Staubli VAL3: FibraHSI.pjx

--- FibraHSI.pjx ---
Parameters version=s7.7.2 stackSize=5000 millimeterUnit=true
Program file=main.pgx
Program file=pLogger.pgx
Program file=start.pgx
Program file=stop.pgx
Program file=usrButtonTxt.pgx
Program file=usrContinue.pgx
Program file=usrSelect.pgx
Data file=FibraHSI.dtx

--- FibraHSI.dtx ---
public frame fFrame = {x=317.444674, y=77.778782, z=-312.57185, rx=-0.864374, ry=0.359034, rz=1.064618, fatherId=world[0]}
public jointRx jJointRx = {j1=45, j2=45, j3=45, j4=45, j5=45, j6=45}
public jointRx jJointRxZeros
public mdesc mMdescFibra = {accel=5, vel=10, decel=5, tmax=10, rmax=10, leave=10, reach=10, blend=cartesian}
public mdesc mMdescMov = {accel=90, decel=90, tmax=99.999, rmax=99.999, blend=cartesian}
mdesc mNomSpeed
num nNumPort = 1000
num nReceiveByte[64]
num nResult
num nXPosButTxt[9]
  [2] = 5
  [3] = 10
  [4] = 15
  [5] = 20
  [6] = 25
  [7] = 30
  [8] = 35
num nYPosButTxt = 13
pointRx pPointRxOrigin = {ry=180, fatherId=fFrame[0]}
pointRx pTempSocket = {fatherId=fFrame[0]}
public sio sSio = {link=Socket\fibra_ser}
public string sInputMsg
public string sOutputMsg
tool ftool = {x=76.72, y=-0.63, z=152.93, fatherId=flange[0], ioLink=valve1}
public tool tTool = {z=20, fatherId=flange[0], ioLink=valve1}
string sOutputMsgLog

--- main.pgx ---
public program main()
  local bool bCom
  local bool bMove
  local bool bOk
  local bool bStop
  local num i
  local num j
  local num nLenMsg
  local num nOffsX
  local num nOffsY
  local num nOverlap
  local num nPosString
  local num nStepX
  local num nStepY
  local num nStepsX
  local num nStepsY
  local num nWhichBttn
  local num nWidthX
  local num nWidthY
  local string sTemp
  local string sXVal
  local string sYVal
  local trsf trsfApproZ20
  local trsf trsfApproZ5
  local trsf trsfTempMove
begin

  userPage()
  cls()
  putln("Please Press F8 to START")
  call usrButtonTxt(8,"HERE")
  //call usrContinue(nWhichBttn, false)
  call usrSelect(nWhichBttn)
  nWhichBttn=-1
  movej(jJointRxZeros,flange,mNomSpeed)
  waitEndMove()

  nNumPort=1000
  sInputMsg=""
  sOutputMsg=""

  sioCtrl(sSio,"port",nNumPort)
  //sioCtrl( sSio, "target",x_sIP)
  sioCtrl(sSio,"endOfString",13)
  sioCtrl(sSio,"nangle",true)
  sioCtrl(sSio,"timeout",0)
  sioCtrl(sSio,"clients",1)

  // If coms or manual aks user or wait Start Comand
  cls()
  putln("Waiting for the 'START' command ...")
  bOk=false
  while bOk==false
    sInputMsg=sSio
    if sInputMsg=="START"
      bOk=true
    else
      bOk=false
    endIf
  endWhile


  // TAREA DE LOGGING
  taskCreate "LoggerTask", 10, pLogger()


  if bOk==true
    // Aproximacion a punto origen Escaneo
    trsfApproZ20={0,0,-20,0,0,0}
    trsfApproZ5={0,0,-5,0,0,0}
    nStepX=0
    nStepY=0

    movej(appro(pPointRxOrigin,trsfApproZ20),tTool,mNomSpeed)
    movel(appro(pPointRxOrigin,trsfApproZ5),tTool,mMdescMov)
    waitEndMove()

    bStop=false
    while bStop==false
      cls()
      putln("Waiting the 'MOVE' / 'STOP' command ...")
      bMove=false
      sInputMsg=sSio
      sTemp=left(sInputMsg,4)
      if sTemp=="MOVE"
        nLenMsg=len(sInputMsg)
        cls()
        putln("Comand Received: "+toString("",nLenMsg))
        putln("   STR: "+sInputMsg)
        putln("   CMD: "+sTemp)
        sTemp=right(sInputMsg,nLenMsg-5)
        putln("   COORD: "+sTemp)
        // Split now the X and Y
        nPosString=find(sTemp,",")
        sXVal=left(sTemp,nPosString)
        nLenMsg=len(sTemp)
        sYVal=right(sTemp,nLenMsg-nPosString-1)
        toNum(sXVal,nStepX,bMove)
        toNum(sYVal,nStepY,bMove)
        putln("   Steps: ")
        putln("      OffsX: "+toString("1.3",nStepX))
        putln("      OffsY: "+toString("1.3",nStepY))
        putln("")
        bMove=true
        //        call usrContinue(nWhichBttn, false)
        //        if nWhichBttn == 8
        //          bMove = true
        //        else
        //          bMove = false
        //        endIf
      elseIf sTemp=="STOP"
        bStop=true
      else
        bMove=false
      endIf

      if bStop==true
        trsfTempMove.z=trsfTempMove.z-20
        movel(appro(pPointRxOrigin,trsfTempMove),tTool,mMdescMov)
        movej(jJointRxZeros,flange,mNomSpeed)
        waitEndMove()
        sOutputMsg="STOPPED"
        sSio=sOutputMsg
        stopMove()
        return
      else
        cls()
      endIf

      if bMove==true
        //Prepare Movement
        trsfTempMove.x=trsfApproZ5.x-nStepX
        trsfTempMove.y=trsfApproZ5.y+nStepY
        // Move robot
        movel(appro(pPointRxOrigin,trsfTempMove),tTool,mMdescFibra)
        waitEndMove()
        pTempSocket=appro(pPointRxOrigin,trsfTempMove)
        sOutputMsg="POS,"+toString("",i)+","+toString("",j)+","+toString(".2",pTempSocket.trsf.x)+","+toString(".2",pTempSocket.trsf.y)
        sSio=sOutputMsg
      else
        sOutputMsg="NOT MOVED"
        // sSio=sOutputMsg
      endIf

    endWhile

    // Return to home
    trsfTempMove.z=trsfTempMove.z-20
    movel(appro(pPointRxOrigin,trsfTempMove),tTool,mMdescMov)
    movej(jJointRxZeros,flange,mNomSpeed)
    waitEndMove()
  else
    stopMove()
    return
  endIf

end

--- start.pgx ---
program start()
begin
  call main()
end

--- pLogger.pgx ---
public program pLogger()
  local joint jHere
  local point pHere
  local num nStart
  local num tEnd
begin
  //Definimos un punto inicial de logging sobre el que computar el tiempo relativo
  nStart=clock()
  //Quizas se pueda iniciar el logging ante una entrada digital que sincronice el laser tracker con el logging.
  while true
    tEnd = clock()-nStart
    sOutputMsgLog = "ts," +toString(".3", tEnd)
    jHere = herej()
    sOutputMsgLog = sOutputMsgLog + ",JOINTS," + toString(".3", jHere.j1) + "," + toString(".3", jHere.j2) + "," + toString(".3", jHere.j3) + "," + toString(".3", jHere.j4) + "," + toString(".3", jHere.j5) + "," + toString(".3", jHere.j6)
    pHere = here(tTool, world)
    sOutputMsgLog = sOutputMsgLog + ",CART,"
    sOutputMsgLog = sOutputMsgLog + toString(".3", pHere.trsf.x) + "," + toString(".3", pHere.trsf.y) + "," + toString(".3", pHere.trsf.z) + ","
    sOutputMsgLog = sOutputMsgLog + toString(".3", pHere.trsf.rx) + "," + toString(".3", pHere.trsf.ry) + "," + toString(".3", pHere.trsf.rz)
    sSio=sOutputMsgLog
    delay(0.02)
  endWhile
end

--- usrButtonTxt.pgx ---
program usrButtonTxt(num x_nWhichButton (dimensions=1), string x_sButtonTxt (dimensions=1))
begin
  //-----------------------------------------------------------------------
  //Header begin
  //Description of program
  //  This program lets you choose the button to display
  //
  //Input parameters
  //  num x_nWhichButton :
  //    role : choice of the navigation key
  //    possible values : 1 to 8 (F1 to F8)
  //
  //  string x_sButtonTxt :
  //    role : Displays desired text
  //
  //Traceability
  //  Creation : 07-04-08 - f.Rob
  //Header end
  //-----------------------------------------------------------------------

  //Position cursor X, Y
  gotoxy(nXPosButTxt[x_nWhichButton],nYPosButTxt)
  //Displays Text
  put(left(x_sButtonTxt,4))
  //Erases contents of  text button parameters
  x_sButtonTxt=" "
end

--- usrContinue.pgx ---
public program usrContinue(num& nWhichBttn (dimensions=1), bool bClear (dimensions=1))
begin
  if bClear
    cls()
    userPage()
    gotoxy(0,0)
    putln("                CONTINUE?")
    call usrButtonTxt(1,"NO")
    call usrButtonTxt(8,"YES")
  else
    putln("                CONTINUE?")
    call usrButtonTxt(1,"NO")
    call usrButtonTxt(8,"YES")
  endIf
  nWhichBttn=-1
  do
    nWhichBttn=(get()-270)
  until ((nWhichBttn==1) or (nWhichBttn==8))
end

--- usrSelect.pgx ---
public program usrSelect(num& nWhichBttn (dimensions=1))
begin
  nWhichBttn=-1
  do
    nWhichBttn=(get()-270)
  until ((nWhichBttn==1) or (nWhichBttn==8))
end
